ABB RobotStudio station: Orange_classification.rspag

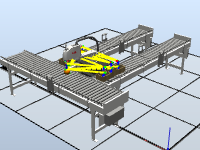
--- station ---
Station Proyectos (saved by RobotStudio 6.8.8307.1040)
Controller Sistema1, task T_ROB1: task frame (RAPID world) sits at (2240.31, -479.99, 843.16) mm, rotated rx 0 ry 0 rz 90.05 deg in the station
Controller Sistema1
  mechanical unit ROB_1: IRB910SC_3_65__01, 4 joints, base frame (0, 0, 0) mm
Layout (positions relative to the parent item):
  - IRB910SC_3_65__01 [mechanism, from Robots\IRB910SC_3_65__01.rslib] at (2240.31, -479.99, 843.16) mm, rotated rx 0 ry 0 rz 90.05 deg; joint values [-0.0882, -0.069, -0.0583, 2.074] (rad or m)
  - 600_guide [part, from Equipment\Conveyor Guide 600.rslib] at (923.39, 0, 0) mm
  - Robotpedestal1400_H240 [part, from Equipment\Robot Pedestal 1400 H240.rslib] at (2217.59, -529.81, 623.95) mm
  - Robotpedestal1400_H240_2 [part, from Equipment\Robot Pedestal 1400 H240.rslib] at (2217.49, -535.49, 419.68) mm
  - Robotpedestal1400_H240_3 [part, from Equipment\Robot Pedestal 1400 H240.rslib] at (2225.5, -527.35, 191.39) mm
  - Robotpedestal1400_H240_4 [part, from Equipment\Robot Pedestal 1400 H240.rslib] at (2226.26, -530.96, -17.61) mm
  - Pieza_6 [part] at (2600.12, -260.63, 769.55) mm
  - 400_guide [part, from Equipment\Conveyor Guide 400.rslib] at (2931.86, -3023.44, -10.63) mm, rotated rx 0 ry 0 rz 90 deg
  - 400_guide_2 [part, from Equipment\Conveyor Guide 400.rslib] at (1841.01, -3030.29, 0) mm, rotated rx 0 ry 0 rz 90 deg
  - Cajita [part] at (1551.06, -265.13, 775.24) mm
  - Cajita_2 [part] at (1555.01, -489.52, 775.57) mm
  - Cajita_3 [part] at (2595.81, -516.34, 777.41) mm
  - Cajita_4 [part] at (1546.3, -709.34, 778.78) mm
  - Cajita_5 [part] at (2599.42, -756.73, 779.01) mm
  - Pieza_8 [part]
  - Attacher_2 [smart component, from Components\Attacher.rslib]
      properties: Parent=IRB910SC_3_65__01; Flange=0; Child=Pieza_8; Mount=false; Offset=[0 0 0]; Orientation=[0 0 0]
  - Detacher [smart component, from Components\Detacher.rslib]
      properties: Child=Pieza_8; KeepPosition=true
  - LogicGate [smart component, from Components\LogicGate.rslib]
      properties: Operator=NOT; Delay=0
  - Positioner [smart component, from Components\Positioner.rslib]
      properties: Object=Pieza_8; Position=[0.6 0 0.015]; Orientation=[0 0 0]; Reference=Global; ReferenceObject=(none)
  - LinearMover [smart component, from Components\LinearMover.rslib]
      properties: Object=Pieza_8; Direction=[-1 0 0]; Speed=0.3; Reference=Global; ReferenceObject=(none)
  - PlaneSensor [smart component, from Components\PlaneSensor.rslib]
      properties: Origin=[2.276378 0.183309 0.82531]; Axis1=[0 0 0.07]; Axis2=[0 0.07 0]; SensedPart=(none)
    - _sensorPart_ [part]
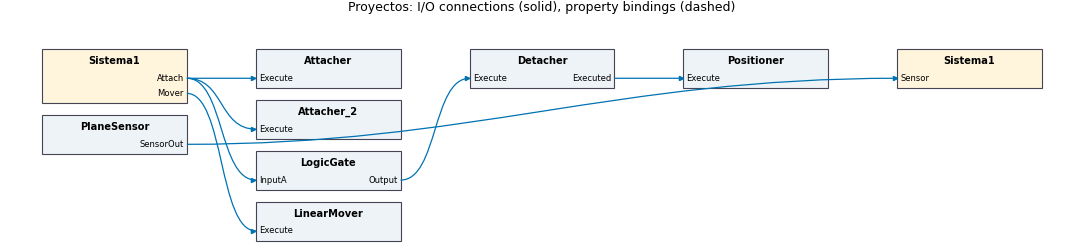
Station logic (signal -> signal, property => property):
  Sistema1.Attach -> Attacher.Execute
  Sistema1.Attach -> Attacher_2.Execute
  Sistema1.Attach -> LogicGate.InputA
  LogicGate.Output -> Detacher.Execute
  Detacher.Executed -> Positioner.Execute
  Sistema1.Mover -> LinearMover.Execute
  PlaneSensor.SensorOut -> Sistema1.Sensor
Targets, tools, work objects and paths stored in the station and not in the controller backup, written as RAPID:
! task T_ROB1
MODULE CalibData
  PERS tooldata Puntita:=[TRUE,[[0,0,0],[1,0,0,0]],[4,[0,0,1],[1,0,0,0],0,0,0]];
  PERS tooldata AloTool:=[TRUE,[[0,0,40],[1,0,0,0]],[0.4,[0,0,1],[1,0,0,0],0,0,0]];
  PERS tooldata MyTool:=[TRUE,[[31.792631019,0,229.638935148],[0.945518576,0,0.325568154,0]],[1,[0,0,1],[1,0,0,0],0,0,0]];
ENDMODULE

! task T_ROB1
MODULE Module1
  CONST robtarget Home:=[[643.95870406,-74.553213185,203.640912982],[0.000422297,0,0,0.999999911],[0,0,0,0],[9E+09,9E+09,9E+09,9E+09,9E+09,9E+09]];
  CONST robtarget Caja1:=[[318.968972197,-460.082866383,-63.609087018],[0.706808109,0,0,-0.707405327],[0,0,0,0],[9E+09,9E+09,9E+09,9E+09,9E+09,9E+09]];
  CONST robtarget Naranja:=[[637.753542427,-85.397976212,37.930912982],[0.706808109,0,0,-0.707405327],[0,0,0,0],[9E+09,9E+09,9E+09,9E+09,9E+09,9E+09]];
ENDMODULE


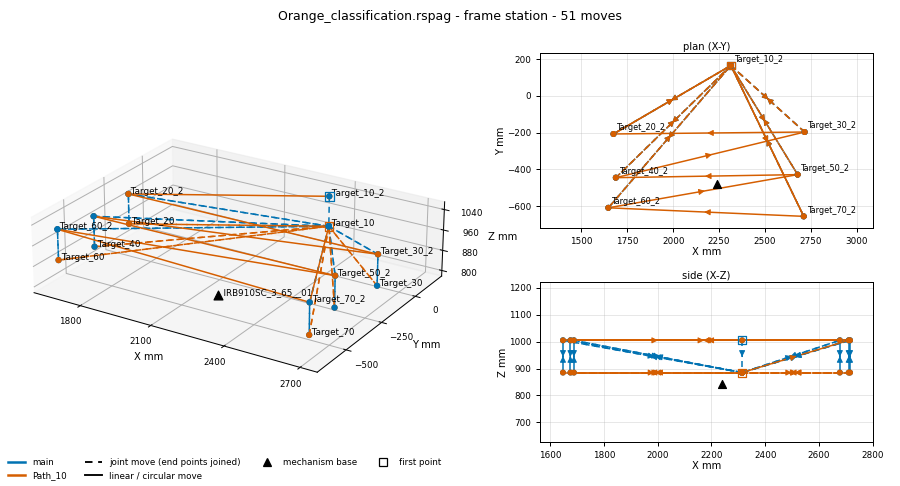
[picture p0: tool path of Orange_classification.rspag in frame station, 51 of 51 moves have a stored position in this frame; points joined in program order, loops and branches not executed]
--- Backups/Sistema1/RAPID/TASK1/PROGMOD/Module1.mod ---
MODULE Module1
	CONST robtarget Target_10:=[[645.361628388,-74.377374159,41.892741812],[0,-0.439613657,0.89818697,0],[-1,1,0,1],[9E+09,9E+09,9E+09,9E+09,9E+09,9E+09]];
	CONST robtarget Target_20:=[[273.164682924,565.04175531,41.892741812],[0,-0.34517174,0.938539541,0],[0,2,0,0],[9E+09,9E+09,9E+09,9E+09,9E+09,9E+09]];
	CONST robtarget Target_30:=[[282.890575697,-475.913992853,41.892741812],[0,0.509754155,0.860320115,0],[-1,2,0,0],[9E+09,9E+09,9E+09,9E+09,9E+09,9E+09]];
	CONST robtarget Target_40:=[[35.242533768,552.520741896,41.892741812],[0,-0.67125191,0.741229299,0],[0,2,0,0],[9E+09,9E+09,9E+09,9E+09,9E+09,9E+09]];
	CONST robtarget Target_50:=[[50.960408769,-437.765098633,41.892741812],[0,0.517953512,0.855408768,0],[-2,2,0,0],[9E+09,9E+09,9E+09,9E+09,9E+09,9E+09]];
	CONST robtarget Target_60:=[[-128.840894088,593.296446909,41.892741812],[0,0.892793921,-0.450465332,0],[0,-2,0,0],[9E+09,9E+09,9E+09,9E+09,9E+09,9E+09]];
	CONST robtarget Target_70:=[[-176.287904502,-470.577490734,41.892741812],[0,-0.534224663,0.84534254,0],[-2,-4,0,0],[9E+09,9E+09,9E+09,9E+09,9E+09,9E+09]];
    CONST robtarget Target_70_2:=[[-176.287904502,-470.577490734,161.892741812],[0,-0.534224663,0.84534254,0],[-2,-4,0,0],[9E+09,9E+09,9E+09,9E+09,9E+09,9E+09]];
    CONST robtarget Target_60_2:=[[-128.840894088,593.296446909,161.892741812],[0,0.892793921,-0.450465332,0],[0,-2,0,0],[9E+09,9E+09,9E+09,9E+09,9E+09,9E+09]];
    CONST robtarget Target_50_2:=[[50.960408769,-437.765098633,161.892741812],[0,0.517953512,0.855408768,0],[-2,2,0,0],[9E+09,9E+09,9E+09,9E+09,9E+09,9E+09]];
    CONST robtarget Target_40_2:=[[35.242533768,552.520741896,161.892741812],[0,-0.67125191,0.741229299,0],[0,2,0,0],[9E+09,9E+09,9E+09,9E+09,9E+09,9E+09]];
    CONST robtarget Target_30_2:=[[282.890575697,-475.913992853,161.892741812],[0,0.509754155,0.860320116,0],[-1,2,0,0],[9E+09,9E+09,9E+09,9E+09,9E+09,9E+09]];
    CONST robtarget Target_20_2:=[[273.164682924,565.04175531,161.892741812],[0,-0.34517174,0.938539541,0],[0,2,0,0],[9E+09,9E+09,9E+09,9E+09,9E+09,9E+09]];
    CONST robtarget Target_10_2:=[[645.361628388,-74.377374159,161.892741812],[0,-0.439613657,0.89818697,0],[-1,1,0,1],[9E+09,9E+09,9E+09,9E+09,9E+09,9E+09]];
    !***********************************************************
    !
    ! Módulo:  Module1
    !
    ! Descripción:
    !   <Introduzca la descripción aquí>
    !
    ! Autor: Carlos Ramos
    !
    ! Versión: 1.0
    !
    !***********************************************************


    !***********************************************************
    !
    ! Procedimiento Main
    !
    !   Este es el punto de entrada de su programa
    !
    !***********************************************************
    PROC main()
        MoveJ Target_10_2,v1000,z100,tool0\WObj:=wobj0;
        SetDO Attach, 0;
        SetDO Mover, 0;
        WaitTime 1;
        MoveJ Target_10,v1000,z100,tool0\WObj:=wobj0;
        WaitTime 1;
        SetDO Attach, 1;
	    MoveJ Target_20_2,v1000,z100,tool0\WObj:=wobj0;
        WaitTime 1;
        MoveJ Target_20,v1000,z100,tool0\WObj:=wobj0;
        WaitTime 1;
        SetDO Attach, 0;
        MoveJ Target_20_2,v1000,z100,tool0\WObj:=wobj0;
        WaitTime 1;

	    MoveJ Target_10,v1000,z100,tool0\WObj:=wobj0;
        SetDO Mover,1;
        WaitDI Sensor, 1;
        SetDO Mover,0;

        WaitTime 1;
        MoveJ Target_10,v1000,z100,tool0\WObj:=wobj0;
        WaitTime 1;
        SetDO Attach, 1;
	    MoveJ Target_30_2,v1000,z100,tool0\WObj:=wobj0;
        WaitTime 1;
        MoveJ Target_30,v1000,z100,tool0\WObj:=wobj0;
        WaitTime 1;
        SetDO Attach, 0;
        MoveJ Target_30_2,v1000,z100,tool0\WObj:=wobj0;
        WaitTime 1;

        MoveJ Target_10,v1000,z100,tool0\WObj:=wobj0;
        SetDO Mover,1;
        WaitDI Sensor, 1;
        SetDO Mover,0;

        WaitTime 1;
        MoveJ Target_10,v1000,z100,tool0\WObj:=wobj0;
        WaitTime 1;
        SetDO Attach, 1;
	    MoveJ Target_70_2,v1000,z100,tool0\WObj:=wobj0;
        WaitTime 1;
        MoveJ Target_70,v1000,z100,tool0\WObj:=wobj0;
        WaitTime 1;
        SetDO Attach, 0;
        MoveJ Target_70_2,v1000,z100,tool0\WObj:=wobj0;
        WaitTime 1;

        MoveJ Target_10,v1000,z100,tool0\WObj:=wobj0;
        SetDO Mover,1;
        WaitDI Sensor, 1;
        SetDO Mover,0;

        WaitTime 1;
        MoveJ Target_10,v1000,z100,tool0\WObj:=wobj0;
        WaitTime 1;
        SetDO Attach, 1;
	    MoveJ Target_50_2,v1000,z100,tool0\WObj:=wobj0;
        WaitTime 1;
        MoveJ Target_50,v1000,z100,tool0\WObj:=wobj0;
        WaitTime 1;
        SetDO Attach, 0;
        MoveJ Target_50_2,v1000,z100,tool0\WObj:=wobj0;
        WaitTime 1;

        MoveJ Target_10,v1000,z100,tool0\WObj:=wobj0;
        SetDO Mover,1;
        WaitDI Sensor, 1;
        SetDO Mover,0;

        WaitTime 1;
        MoveJ Target_10,v1000,z100,tool0\WObj:=wobj0;
        WaitTime 1;
        SetDO Attach, 1;
	    MoveJ Target_40_2,v1000,z100,tool0\WObj:=wobj0;
        WaitTime 1;
        MoveJ Target_40,v1000,z100,tool0\WObj:=wobj0;
        WaitTime 1;
        SetDO Attach, 0;
        MoveJ Target_40_2,v1000,z100,tool0\WObj:=wobj0;
        WaitTime 1;

        MoveJ Target_10,v1000,z100,tool0\WObj:=wobj0;
        SetDO Mover,1;
        WaitDI Sensor, 1;
        SetDO Mover,0;

        WaitTime 1;
        MoveJ Target_10,v1000,z100,tool0\WObj:=wobj0;
        WaitTime 1;
        SetDO Attach, 1;
	    MoveJ Target_60_2,v1000,z100,tool0\WObj:=wobj0;
        WaitTime 1;
        MoveJ Target_60,v1000,z100,tool0\WObj:=wobj0;
        WaitTime 1;
        SetDO Attach, 0;
        MoveJ Target_60_2,v1000,z100,tool0\WObj:=wobj0;
        WaitTime 1;

        MoveJ Target_10,v1000,z100,tool0\WObj:=wobj0;
        SetDO Mover,1;
        WaitDI Sensor, 1;
        SetDO Mover,0;
    ENDPROC
	PROC Path_10()
	    MoveJ Target_10,v1000,z100,tool0\WObj:=wobj0;
	    MoveJ Target_20,v1000,z100,tool0\WObj:=wobj0;
	    MoveJ Target_10,v1000,z100,tool0\WObj:=wobj0;
	    MoveJ Target_30,v1000,z100,tool0\WObj:=wobj0;
	    MoveJ Target_10,v1000,z100,tool0\WObj:=wobj0;
	    MoveJ Target_40,v1000,z100,tool0\WObj:=wobj0;
	    MoveJ Target_10,v1000,z100,tool0\WObj:=wobj0;
	    MoveJ Target_50,v1000,z100,tool0\WObj:=wobj0;
	    MoveJ Target_10,v1000,z100,tool0\WObj:=wobj0;
	    MoveJ Target_60,v1000,z100,tool0\WObj:=wobj0;
	    MoveJ Target_10,v1000,z100,tool0\WObj:=wobj0;
	    MoveJ Target_70,v1000,z100,tool0\WObj:=wobj0;
	    MoveJ Target_10,v1000,z100,tool0\WObj:=wobj0;
        MoveL Target_70_2,v1000,z100,tool0\WObj:=wobj0;
        MoveL Target_60_2,v1000,z100,tool0\WObj:=wobj0;
        MoveL Target_50_2,v1000,z100,tool0\WObj:=wobj0;
        MoveL Target_40_2,v1000,z100,tool0\WObj:=wobj0;
        MoveL Target_30_2,v1000,z100,tool0\WObj:=wobj0;
        MoveL Target_20_2,v1000,z100,tool0\WObj:=wobj0;
        MoveL Target_10_2,v1000,z100,tool0\WObj:=wobj0;
	ENDPROC
ENDMODULE

--- Backups/Sistema1/SYSPAR/EIO.cfg ---
EIO:CFG_1.0:6:1::
#
EIO_SIGNAL:

      -Name "Attach" -SignalType "DO"

      -Name "Mover" -SignalType "DO"

      -Name "Sensor" -SignalType "DI"
